FUNCTION_BLOCK FB_ProtectRelay_WIP1 EXTENDS FB_ProtectRelay_Base
VAR_INPUT
						
	
	

END_VAR

VAR_INPUT
	// I/O Inputs 		                                     				
		IN_MesAlarmImax_IO		: BOOL ; // IO max I  fault
		IN_MesAlarmUmin_IO		: BOOL ;  // IO Min U  Fault 
		
END_VAR


VAR
// M_ALARMMNGMT VARIABLES //
                            		
	CmdResetHVCell				: BOOL ; 
	// M_READ VARIABLES//
	
MesDataExd 		    AT %Q*  	: ProtectRelay_WIP1; 	
		


END_VAR

METHOD M_Execute
SUPER^.M_Execute();
END_METHOD

END_FUNCTION_BLOCK

(* stored: Version 1.1.0.1, ProductVersion 3.1.4024.6
   POU FB_ProtectRelay_WIP1: Id {4760cdfe-8439-4d6a-b69e-cc968374b761}, SpecialFunc None
   Method M_Execute: Id {a741c423-9032-47eb-9598-a4dcd1713ad3} *)
